Yaskawa INFORM job: POS_WORKPIECE.JBI

/JOB
//NAME POS_WORKPIECE
///FOLDERNAME INNE
//POS
///NPOS 6,6,0,0,0,0
///TOOL 0
///POSTYPE PULSE
///PULSE
C00000=-107372,-15205,-22015,22157,89921,46116
C00001=-142764,-7201,-14847,21973,99256,34902
C00002=-73784,22583,11442,18465,80407,56600
C00003=106930,-26869,-30362,-22128,89011,-46118
C00004=145066,-20338,-24755,-21750,99265,-34059
C00005=71287,11466,1263,-18023,80391,-57500
BC00000=148911,121620,531712
BC00001=148911,121619,531709
BC00002=148911,121619,531709
BC00003=148911,121619,531709
BC00004=148911,121619,531707
BC00005=148911,121619,531707
//INST
///DATE 2023/10/04 15:16
///ATTR SC,RW
///GROUP1 RB1,BS1
NOP
MOVJ C00000 BC00000 VJ=0.78 PL=0
MOVJ C00001 BC00001 VJ=0.78 PL=0
MOVJ C00002 BC00002 VJ=0.78 PL=0
MOVJ C00003 BC00003 VJ=0.78 PL=0
MOVJ C00004 BC00004 VJ=0.78 PL=0
MOVJ C00005 BC00005 VJ=0.78 PL=0
END
